// TIA Portal V19 export
DATA_BLOCK "SINA_SPEED_TLG352_DB"   // DB37
AUTHOR : SIEMENS
FAMILY : DRIVES
NAME : SINA_SPD_TLG352
VERSION : 1.0
// stored: InstanceOfName SINA_SPEED_TLG352, InstanceOfType FB
"SINA_SPEED_TLG352"
   // VAR_INPUT
   //    enableAxis : Bool;
   //    ackError : Bool;
   //    speedSp : Real;
   //    userPZD1 : Word;
   //    userPZD2 : Word;
   //    userPZD3 : Word;
   //    userPZD4 : Word;
   //    refSpeed : Real;
   //    refCurrent : Real;
   //    refTorque : Real;
   //    configAxis : Word;
   //    HWIDSTW : HW_IO;
   //    HWIDZSW : HW_IO;
   // END_VAR
   // VAR_OUTPUT
   //    axisEnabled : Bool;
   //    lockout : Bool;
   //    actSpeed : Real;
   //    actCurrent : Real;
   //    actTorque : Real;
   //    warnCode : UInt;
   //    faultCode : UInt;
   //    error : Bool;
   //    status : Int;
   //    diagId : Int;
   // END_VAR
BEGIN
END_DATA_BLOCK
